// TIA Portal V19 export
DATA_BLOCK "_IOL_VM_TPV50-9_Params"   // DB503
TITLE = Valve Monitoring Params for Tetra Pak V50 DeviceID: 9
{ S7_Optimized_Access := 'TRUE' }
// stored: AutoNumber false, MemoryReserve 0
   VAR RETAIN
      VM_IOL_Params : "_IOL_VM_TPV50_9";
   END_VAR
BEGIN
   VM_IOL_Params.StandardStructure.Parameter3.Subindex := 0;
END_DATA_BLOCK
